FUNCTION_BLOCK FB_ST10
VAR
	_Camera : BOOL;
	_Scanner : BOOL;
	_triger : BOOL;
	_busy  : BOOL;
	_desc : STRING;
END_VAR

METHOD PROTECTED _camera
VAR_INPUT
END_VAR
IF _Camera THEN 
	_desc:= 'Camera ready';
ELSIF _triger THEN 
	_desc:= 'Triger';
ELSE
	_busy:= FALSE;
END_IF
END_METHOD

END_FUNCTION_BLOCK

(* stored: Version 1.1.0.1, ProductVersion 3.1.4024.12
   POU FB_ST10: Id {69545744-4ffd-44e8-84c0-cbb5f2cc935d}, SpecialFunc None
   Method _camera: Id {0be8627e-1fb1-44dc-8173-3e82e3599b26} *)
